TYPE
    ST_HMI_ControlInPut :
    STRUCT
        Input  : ST_InputTables;
        Output : ST_OutputTables;
    END_STRUCT
END_TYPE

(* stored: Version 1.1.0.1, ProductVersion 3.1.4024.13
   DUT ST_HMI_ControlInPut: Id {707bb554-82de-4df0-bd0f-e5b009bdf722} *)
